FUNCTION_BLOCK Z_CONTROLLER (* Basic FB with empty ECC *)
  (* Standard: 61499-2 *)
  (* Version 1.0, 2020-10-18, chong *)
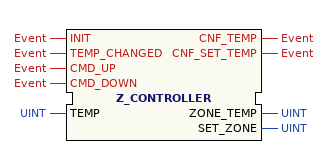
  EVENT_INPUT
    INIT;
    TEMP_CHANGED;
    CMD_UP;
    CMD_DOWN;
  END_EVENT
  EVENT_OUTPUT
    CNF_TEMP;
    CNF_SET_TEMP;
  END_EVENT
  VAR_INPUT
    TEMP : UINT;
  END_VAR
  VAR_OUTPUT
    ZONE_TEMP : UINT;
    SET_ZONE : UINT;
  END_VAR
  EC_STATES
    START; (* Initial State *)
  END_STATES
END_FUNCTION_BLOCK
